FUNCTION_BLOCK Potentiometer
VAR
	nInput	AT%I*	: INT;
END_VAR

PROPERTY ActualValue : INT
GET
ActualValue := nInput;
END_GET
END_PROPERTY

PROPERTY ActualValuePercent : LREAL
GET
ActualValuePercent := F_Scale ( nInput, 0, 32767, 0, 100 );
END_GET
END_PROPERTY

END_FUNCTION_BLOCK

(* stored: Version 1.1.0.1
   POU Potentiometer: Id {a084b3b6-26cc-4a31-8637-da3898d58a44}, SpecialFunc None
   Property ActualValue: Id {c8135842-bb71-4358-8401-9fdd5fc3256a}
   Get Get: Id {7599e485-e8fa-4b6d-9a83-672ac6f443b8}
   Property ActualValuePercent: Id {35661c7a-00e3-4b0a-b66e-16f51f6800bb}
   Get Get: Id {3900818d-9e8c-4148-847c-8ddf98549df6} *)
